(* CODESYS project bargeControl
   Author: Sigurd Rød Brekk
   Company: ScaleAQ
   Description: Control and monitoring of processe related to the barges.
   Title: bargeControl
   Version: 0.0.0

Project tree, tasks and I/O mapping:
  PFC100_Simulation : 750-8111 PFC100, WAGO, order no. 750-8111, version 6.2.0.1
    application Application
      libraries: Standard, 3.5.18.0 (System); WagoSysDynamicIoMapping, 1.0.4.0 (WAGO); SysTask, * (System)
      task BilgePump (cyclic, interval 100 ms, priority 1, watchdog 20 ms x 1) calls BilgePump
      task IOSimulation (cyclic, interval 100 ms, priority 1, watchdog 20 ms x 1) calls simulationMapping
      task TankLevel (cyclic, interval 100 ms, priority 1, watchdog 20 ms x 1) calls TankLevel
      GVL/
        global variables GVL_Simulation
      global variables PersistentVars
      program simulationMapping [ST]
      Symbols
    Kbus : Kbus, WAGO, version 2.1.0.1
        unmapped channels: K-BUS diagnostics
  SiteProgram : 750-8111 PFC100, WAGO, order no. 750-8111, version 6.2.0.1
    application Application
      libraries: Standard, 3.5.18.0 (System); WagoSysDynamicIoMapping, 1.0.4.0 (WAGO); SysTask, * (System)
      task BilgePump (cyclic, interval 100 ms, priority 2, watchdog 20 ms x 1) calls BilgePump
      task ReadIOCards (cyclic, interval 100 ms, priority 1, watchdog 20 ms x 1) calls DynamicIOConfig, ReadInputs
      task TankLevel (cyclic, interval 100 ms, priority 14, watchdog 20 ms x 1) calls TankLevel
      task WriteIOCards (cyclic, interval 100 ms, priority 15, watchdog 20 ms x 1) calls WriteOutputs
      GVL/
        global variables GVL_WagoIO
      global variables PersistentVars
      PRG/
        program DynamicIOConfig [ST]
        program ReadInputs [ST]
        program WriteOutputs [ST]
      Symbols
    Kbus : Kbus, WAGO, version 2.1.0.1
        unmapped channels: K-BUS diagnostics
  SoftSimulation : CODESYS Control Win V3 x64, 3S - Smart Software Solutions GmbH, version 3.5.19.50
    application Application
      libraries: Standard, 3.5.18.0 (System); SysTask, * (System)
      task BilgePump (cyclic, interval 100 ms, priority 1, watchdog 20 ms x 1) calls BilgePump
      task IOSimulation (cyclic, interval 100 ms, priority 1, watchdog 20 ms x 1) calls simulationMapping
      task TankLevel (cyclic, interval 100 ms, priority 1, watchdog 20 ms x 1) calls TankLevel
      task TrendRecordingTask (cyclic, interval 100 ms, priority 31) calls VisuTrendStorageAccess.GlobalInstances.g_TrendRecordingManager.CyclicCall
      task VISU_TASK (cyclic, interval 100 ms, priority 31) calls VisuElems.Visu_Prg
      global variables GVL_Simulation
      global variables PersistentVars
      program simulationMapping [ST]
      Symbols
      Trend Recording Manager
        TrendRecording
      visualisation Visualization
  ENUM/
    data type AlarmState
    data type powerState
    data type tankShape
    data type unitType
  FB/
    function block AlarmManagement [ST]
    function block BilgeControl [ST]
    function block Butterworth [ST]
  FUNCTION/
    function analogInputToMeter [ST]
    function heightToVolume [ST]
  text list GlobalTextList
  GVL/
    global variables GVL_IO
    global variables GVL_Retain
    global variables GVL_UPS
  PRG/
    program BilgePump [ST]
    program TankLevel [ST]
  STRUCT/
    data type AlarmStructBilge
    data type AlarmStructTankLevel
    data type BilgeObject
    data type IOSetup
    data type PowerSupply
    data type TankLevelObject
    data type UPS
*)

// ENUM/AlarmState
{attribute 'qualified_only'}
{attribute 'strict'}
TYPE AlarmState :
(
	Normal,
	UnacknowledgedAlarm,
	AcknowledgedAlarm,
	RTNunacknowledged
);
END_TYPE

// ENUM/powerState
{attribute 'qualified_only'}
{attribute 'strict'}
TYPE powerState :
(
	normal,
	noVoltage,
	fuseBlown
);
END_TYPE

// ENUM/tankShape
{attribute 'qualified_only'}
{attribute 'strict'}
TYPE tankShape :
(
	notDefined,
	rectangle,
	cylindrical
);
END_TYPE

// ENUM/unitType
{attribute 'qualified_only'}
{attribute 'strict'}
TYPE unitType :
(
	bar,
	meter
);
END_TYPE

// STRUCT/AlarmStructBilge
TYPE AlarmStructBilge :
STRUCT
	waterAlarmState				: AlarmState;
	acknowledgeWaterDetAlm		: BOOL;
	dieselAlarmState			: AlarmState;
	acknowledgeDieselDetAlm		: BOOL;
	manualStartAlarmState		: AlarmState;
	acknowledgeManualStartAlm	: BOOL;
END_STRUCT
END_TYPE

// STRUCT/AlarmStructTankLevel
TYPE AlarmStructTankLevel :
STRUCT
	LAL						: AlarmState;
	acknowledgeLAL			: BOOL;
	LAH						: AlarmState;
	acknowledgeLAH			: BOOL;
	outOfRange				: AlarmState;
	acknowledgeoutOfRange	: BOOL;
END_STRUCT
END_TYPE

// STRUCT/BilgeObject
TYPE BilgeObject :
STRUCT
	available				: BOOL;
	enable					: BOOL;
	auto					: BOOL;
	startManual				: BOOL;
	leakageDetected			: BOOL;
	dieselDetected			: BOOL;
	activateDieselDetection	: BOOL;
	startPump				: BOOL;
	Alarm					: AlarmStructBilge;
END_STRUCT
END_TYPE

// STRUCT/IOSetup
TYPE IOSetup :
STRUCT
	availableBilgeInputs	: INT;
	availableBilgeOutputs	: INT;
	availableAnalogInputs	: INT;
	IOFault					: BOOL;
END_STRUCT
END_TYPE

// STRUCT/PowerSupply
TYPE PowerSupply :
STRUCT
	available	: BOOL;
	state		: powerState;
END_STRUCT
END_TYPE

// STRUCT/TankLevelObject
TYPE TankLevelObject :
STRUCT
	available			: BOOL; //Checks if IO is available in K-BUS
	enable				: BOOL; //Enabled from SiteControl
	engRangeMin			: REAL; //Range on instrument [bar]
	engRangeMax 		: REAL; //Range on instrument [bar]
	rawInput 			: WORD; //input WORD from AD-converter
	filteredInput		: REAL; //filtered input WORD (low pass filter)
	density				: REAL; //density for liquid [kg/m^3]
	levelHeightOuput	: REAL; //height of liquid column [m]
	levelVolumeOutput	: REAL; //Volume [litre]
	tankShape			: tankShape;
	tankparameter		: ARRAY [1..2] OF REAL;
	SetPointLAL			: REAL; //[m]
	SetPointLAH			: REAL; //[m]
	Alarm				: AlarmStructTankLevel;
END_STRUCT
END_TYPE

// STRUCT/UPS
TYPE UPS :
STRUCT
	batteryHealthy	: BOOL;
	mainsConnected	: BOOL;
END_STRUCT
END_TYPE

// GVL/GVL_IO
{attribute 'qualified_only'}
VAR_GLOBAL	
	availableIO			: IOSetup;
END_VAR

// GVL/GVL_Retain
{attribute 'qualified_only'}
VAR_GLOBAL PERSISTENT RETAIN
	bilgePumpArray	: ARRAY [1..28] OF BilgeObject;
	tankLevelArray		: ARRAY [1..12] OF TankLevelObject;
END_VAR

// GVL/GVL_UPS
{attribute 'qualified_only'}
VAR_GLOBAL
	ups : UPS;
END_VAR

// PFC100_Simulation/Application/PersistentVars
{attribute 'qualified_only'}
VAR_GLOBAL PERSISTENT RETAIN
	// Generated instance path of persistent variable
	__POOL.GVL_Retain.bilgePumpArray: ARRAY [1..28] OF BilgeObject;
	// Generated instance path of persistent variable
	__POOL.GVL_Retain.tankLevelArray: ARRAY [1..12] OF TankLevelObject;
END_VAR

// SiteProgram/Application/PersistentVars
{attribute 'qualified_only'}
VAR_GLOBAL PERSISTENT RETAIN
	// Generated instance path of persistent variable
	__POOL.GVL_Retain.bilgePumpArray: ARRAY [1..28] OF BilgeObject;
	// Generated instance path of persistent variable
	__POOL.GVL_Retain.tankLevelArray: ARRAY [1..12] OF TankLevelObject;
END_VAR

// SoftSimulation/Application/GVL_Simulation
{attribute 'qualified_only'}
VAR_GLOBAL
tankLevelSim	: ARRAY [1..12] OF WORD;
bilgeLimitSwitch	: ARRAY [1..28] OF BOOL;
bilgePumpStart		: ARRAY [1..28] OF BOOL;
END_VAR

// SoftSimulation/Application/PersistentVars
{attribute 'qualified_only'}
VAR_GLOBAL PERSISTENT RETAIN
	// Generated instance path of persistent variable
	__POOL.GVL_Retain.bilgePumpArray: ARRAY [1..28] OF BilgeObject;
	// Generated instance path of persistent variable
	__POOL.GVL_Retain.tankLevelArray: ARRAY [1..12] OF TankLevelObject;
END_VAR

// PFC100_Simulation/Application/GVL/GVL_Simulation
{attribute 'qualified_only'}
VAR_GLOBAL
tankLevelSim	: ARRAY [1..12] OF WORD;
bilgeLimitSwitch	: ARRAY [1..28] OF BOOL;
bilgePumpStart		: ARRAY [1..28] OF BOOL;
END_VAR

// SiteProgram/Application/GVL/GVL_WagoIO
{attribute 'qualified_only'}
VAR_GLOBAL
	digitalInputCollection	: ARRAY [1..3] OF WagoSysDynamicIoMapping.I_Module;
	digitalOutputCollection	: ARRAY [1..3] OF WagoSysDynamicIoMapping.I_Module;
	analogInputCollection	: ARRAY [1..3] OF WagoSysDynamicIoMapping.I_Module;
	
END_VAR

// PRG/BilgePump
PROGRAM BilgePump
VAR
	i	: INT;
	BilgeControlArray	: ARRAY[1..28] OF BilgeControl;
	BilgeAlarm			: ARRAY[1..28] OF AlarmManagement;
END_VAR

FOR i := 1 TO 28 DO 
	IF (GVL_Retain.bilgePumpArray[i].available AND GVL_Retain.bilgePumpArray[i].enable) THEN
		BilgeControlArray[i](
			//INPUTS
			leakageDetected			:= GVL_Retain.bilgePumpArray[i].leakageDetected,
			dieselDetected			:= GVL_Retain.bilgePumpArray[i].dieselDetected,
			activateDieselDetection	:= GVL_Retain.bilgePumpArray[i].activateDieselDetection,
			auto					:= GVL_Retain.bilgePumpArray[i].auto,
			startManual				:= GVL_Retain.bilgePumpArray[i].startManual,
			
			//OUTPUTS
			startPump				=> GVL_Retain.bilgePumpArray[i].startPump
		);
		
		//Alarm management	
		//Alarm state for water detection
		BilgeAlarm[i](
			AbnormalCondition		:= GVL_Retain.bilgePumpArray[i].leakageDetected,
			Acknowledge				:= GVL_Retain.bilgePumpArray[i].Alarm.acknowledgeWaterDetAlm,
			ProcessAlarmState		:= GVL_Retain.bilgePumpArray[i].Alarm.waterAlarmState,
		);
		//Alarm state for disel detection
		BilgeAlarm[i](
			AbnormalCondition		:= GVL_Retain.bilgePumpArray[i].dieselDetected,
			Acknowledge				:= GVL_Retain.bilgePumpArray[i].Alarm.acknowledgeDieselDetAlm,
			ProcessAlarmState		:= GVL_Retain.bilgePumpArray[i].Alarm.dieselAlarmState,
		);
		//Alarm state for manual start
		BilgeAlarm[i](
			AbnormalCondition		:= GVL_Retain.bilgePumpArray[i].startManual,
			Acknowledge				:= GVL_Retain.bilgePumpArray[i].Alarm.acknowledgeManualStartAlm,
			ProcessAlarmState		:= GVL_Retain.bilgePumpArray[i].Alarm.manualStartAlarmState,
		);
	ELSE
		GVL_Retain.bilgePumpArray[i].startPump := FALSE;
	END_IF
END_FOR

END_PROGRAM

// FB/BilgeControl
FUNCTION_BLOCK BilgeControl
VAR_INPUT
	leakageDetected			: BOOL;
	dieselDetected			: BOOL;
	activateDieselDetection	: BOOL;
	auto					: BOOL;
	startManual				: BOOL;
END_VAR
VAR_OUTPUT
	startPump				: BOOL;
END_VAR
VAR
	pumpHysteresis	:	TOF;
END_VAR

IF auto THEN
	pumpHysteresis(IN := leakageDetected,PT := T#60S);
	IF (NOT(activateDieselDetection AND dieselDetected) AND leakageDetected) THEN // Only activate bilge pump if diesel is not detected (while activated).
		startPump := pumpHysteresis.Q;
	ELSE 
		startPump := FALSE;
	END_IF
ELSE
	IF startManual THEN
		startPump := TRUE;
	ELSE
		startPump := FALSE;
	END_IF
END_IF

END_FUNCTION_BLOCK

// FB/AlarmManagement
FUNCTION_BLOCK AlarmManagement
VAR_INPUT
	AbnormalCondition	: BOOL;
	Acknowledge			: BOOL;
END_VAR
VAR_IN_OUT
	ProcessAlarmState			: AlarmState;
END_VAR

CASE ProcessAlarmState OF
			0:
				//NORMAL OPERATION
				IF AbnormalCondition THEN
					ProcessAlarmState := 1;
				END_IF
			1:
				//UNACKNOWLEDGED ALARM
				IF NOT AbnormalCondition THEN
					ProcessAlarmState := 3;
				END_IF
				IF Acknowledge THEN
					ProcessAlarmState := 2;
				END_IF
			2:	
				//ACKNOWLEDGED ALARM
				IF NOT AbnormalCondition THEN
					ProcessAlarmState := 0;
				END_IF
			3:
			
				//RTN unacknowledged
				IF AbnormalCondition THEN
					ProcessAlarmState := 1;
				END_IF
				IF Acknowledge THEN
					ProcessAlarmState := 0;
				END_IF
		END_CASE

END_FUNCTION_BLOCK

// PFC100_Simulation/Application/simulationMapping
PROGRAM simulationMapping
VAR
	i	: INT;
	filter				: ARRAY[1..12] OF Butterworth; // second order butterworth filter 
END_VAR

//READ DIGITAL INPUTS FROM IO-CARD
FOR i := 1 TO 28 DO 
	IF (GVL_Retain.bilgePumpArray[i].available AND GVL_Retain.bilgePumpArray[i].enable) THEN
		GVL_Retain.bilgePumpArray[i].leakageDetected := GVL_Simulation.bilgeLimitSwitch[i];
	END_IF
END_FOR

FOR i	:= 1 TO 12 DO
	IF (GVL_Retain.tankLevelArray[i].available AND GVL_Retain.tankLevelArray[i].enable) THEN
	GVL_Retain.tankLevelArray[i].rawInput := GVL_Simulation.tankLevelSim[i];
	//Filter input signal
	filter[i](fc := 0.01, u_in:= GVL_Retain.tankLevelArray[i].rawInput, y_out => GVL_Retain.tankLevelArray[i].filteredInput);
	END_IF
END_FOR

IF (GVL_Retain.bilgePumpArray[i].available AND GVL_Retain.bilgePumpArray[i].enable) THEN
	GVL_Simulation.bilgePumpStart[i] := GVL_Retain.bilgePumpArray[i].startPump;
END_IF

END_PROGRAM

// SoftSimulation/Application/simulationMapping
PROGRAM simulationMapping
VAR
	i	: INT;
	filter				: ARRAY[1..12] OF Butterworth; // second order butterworth filter 
END_VAR

//READ DIGITAL INPUTS FROM IO-CARD
FOR i := 1 TO 28 DO 
	IF (GVL_Retain.bilgePumpArray[i].available AND GVL_Retain.bilgePumpArray[i].enable) THEN
		GVL_Retain.bilgePumpArray[i].leakageDetected := GVL_Simulation.bilgeLimitSwitch[i];
	END_IF
END_FOR

FOR i	:= 1 TO 12 DO
	IF (GVL_Retain.tankLevelArray[i].available AND GVL_Retain.tankLevelArray[i].enable) THEN
	GVL_Retain.tankLevelArray[i].rawInput := GVL_Simulation.tankLevelSim[i];
	//Filter input signal
	filter[i](fc := 0.01, u_in:= GVL_Retain.tankLevelArray[i].rawInput, y_out => GVL_Retain.tankLevelArray[i].filteredInput);
	END_IF
END_FOR

IF (GVL_Retain.bilgePumpArray[i].available AND GVL_Retain.bilgePumpArray[i].enable) THEN
	GVL_Simulation.bilgePumpStart[i] := GVL_Retain.bilgePumpArray[i].startPump;
END_IF

END_PROGRAM

// FB/Butterworth
FUNCTION_BLOCK Butterworth
VAR_INPUT
	fc		: REAL; //cut-off frequency
	u_in	: WORD; //filter input
END_VAR
VAR_OUTPUT
	y_out	: REAL; //filter output
END_VAR
VAR
	yk		: REAL := 0;
	ykm1	: REAL := 0;
	ykm2	: REAL := 0;
	uk		: REAL := 0;
	ukm1	: REAL	:= 0;
	ukm2	: REAL	:= 0;
	//TEST
	hTask:       SysTask.RTS_IEC_HANDLE; // task handle
	Tsu		: UDINT; // interval in micro seconds
	fsample		: REAL;
	fs			: REAL;
	
	A_2		: REAL;
	B_0		: REAL;
	B_1		: REAL;
	B_2		: REAL;
	
	N0		: REAL;
	N1		: REAL;
	N2		: REAL;
	D0		: REAL;
	D1		: REAL;
	D2		: REAL;
END_VAR

SysTaskGetCurrent(ADR(hTask));
SysTaskGetInterval(hTask, Tsu);
fsample := 1000000/(UDINT_TO_REAL(Tsu));
fs := 2*TAN(3.1415926536*((fc)/(fsample)));


uk 		:= WORD_TO_REAL(u_in);

A_2 := LREAL_TO_REAL(EXPT(2*3.1415926536*fs,2));
B_0 := 1;
B_1 := LREAL_TO_REAL(SQRT(2));
B_2 := A_2;

N0 := A_2;
N1 := 2*(A_2);
N2 := A_2;
D0 := B_2 + 2*fs*B_1 + 4*LREAL_TO_REAL(EXPT(fs,2))*B_0;
D1 := 2*(B_2 - 4*LREAL_TO_REAL(EXPT(fs,2))*B_0);
D2 := B_2 - 2*fs*B_1 + 4*LREAL_TO_REAL(EXPT(fs,2))*B_0;




yk		:= ((((N0)/(D0))/1) * (1*uk + ((N1)/(N0))*ukm1 + ((N2)/(N0))*ukm2)) - ((((D1)/(D0))*ykm1+((D2)/(D0))*ykm2));

ykm2 	:= ykm1;
ykm1 	:= yk;

ukm2	:= ukm1;
ukm1	:= uk;

y_out 	:= WORD_TO_REAL(REAL_TO_WORD(yk));

END_FUNCTION_BLOCK

// PRG/TankLevel

PROGRAM TankLevel
VAR
	i	: INT;
	TankAlarm			: ARRAY[1..12] OF AlarmManagement;

	//Alarm conditions
	fluidHigh			: BOOL;
	fluidLow			: BOOL;
	signalFault			: BOOL;
	
END_VAR

FOR i := 1 TO 12 DO 
	IF (GVL_Retain.tankLevelArray[i].available AND GVL_Retain.tankLevelArray[i].enable) THEN
		//Calculate level hegiht
		GVL_Retain.tankLevelArray[i].levelHeightOuput := analogInputToMeter(
			fluidDensity	:= GVL_Retain.tankLevelArray[i].density,
			engRangeMin		:= GVL_Retain.tankLevelArray[i].engRangeMin,
			engRangeMax		:= GVL_Retain.tankLevelArray[i].engRangeMax,
			input			:= GVL_Retain.tankLevelArray[i].filteredInput
		);
		//CALCULATE VOLUME IF DEFINED
		GVL_Retain.tankLevelArray[i].levelVolumeOutput := heightToVolume(
			GVL_Retain.tankLevelArray[i].levelHeightOuput,
			GVL_Retain.tankLevelArray[i].tankShape, 
			GVL_Retain.tankLevelArray[i].tankparameter);
		
		//CHECK IF LEVEL IS BELOW SET POINT FOR LAL
		IF (GVL_Retain.tankLevelArray[i].levelHeightOuput < GVL_Retain.tankLevelArray[i].SetPointLAL) AND (GVL_Retain.tankLevelArray[i].SetPointLAL > 0)  THEN
			fluidLow := TRUE;
		ELSE
			fluidLow := FALSE;
		END_IF
		//CHECK IF LEVEL IS ABOVE SET POINT FOR LAH
		IF (GVL_Retain.tankLevelArray[i].levelHeightOuput > GVL_Retain.tankLevelArray[i].SetPointLAH) AND (GVL_Retain.tankLevelArray[i].SetPointLAH > 0)  THEN
			fluidHigh := TRUE;
		ELSE
			fluidHigh := FALSE;
		END_IF
		//CHECK IF TRANSMITTER VALUE IS OUT OF RANGE - Analog input gives the value 3 if the current is < 3mA, and 32767 if current > 21mA
		IF (GVL_Retain.tankLevelArray[i].rawInput = 3) OR (GVL_Retain.tankLevelArray[i].rawInput = 32767)  THEN
			signalFault := TRUE;
		ELSE
			signalFault := FALSE;
		END_IF
		
		//ALARM MANAGEMENT
		//Alarm state for low level
		TankAlarm[i](
			AbnormalCondition		:= fluidLow,
			Acknowledge				:= GVL_Retain.tankLevelArray[i].Alarm.acknowledgeLAL,
			ProcessAlarmState		:= GVL_Retain.tankLevelArray[i].Alarm.LAL
		);
		//Alarm state for high level
		TankAlarm[i](
			AbnormalCondition		:= fluidHigh,
			Acknowledge				:= GVL_Retain.tankLevelArray[i].Alarm.acknowledgeLAH,
			ProcessAlarmState		:= GVL_Retain.tankLevelArray[i].Alarm.LAH
		);
		//Alarm state for transmitter out of range
		TankAlarm[i](
			AbnormalCondition		:= signalFault,
			Acknowledge				:= GVL_Retain.tankLevelArray[i].Alarm.acknowledgeoutOfRange,
			ProcessAlarmState		:= GVL_Retain.tankLevelArray[i].Alarm.outOfRange
		);
	END_IF
END_FOR

END_PROGRAM

// FUNCTION/analogInputToMeter
FUNCTION analogInputToMeter : REAL //in meters
VAR_INPUT
	fluidDensity		: REAL; //kg/m^3
	engRangeMin			: REAL; // bar
	engRangeMax			: REAL; // bar
	input				: REAL;
END_VAR
VAR
	g					: REAL := 9.8; //[m/s^2]
	res					: REAL := 4095;//analog input resolution
END_VAR

//h = (P)/(rho * g)
IF (fluidDensity > 0) THEN
	analogInputToMeter := ((input*(engRangeMax-engRangeMin)/res)*100000)/(fluidDensity*g);
ELSE
	 analogInputToMeter := 0;
END_IF

END_FUNCTION

// FUNCTION/heightToVolume
FUNCTION heightToVolume : REAL
VAR_INPUT
	height		: REAL;
	shape		: tankShape;
	parameters	: ARRAY [1..2] OF REAL;
END_VAR
VAR
	pi	: REAL := 3.141592653589793238462;
END_VAR

CASE shape OF
			1:
				heightToVolume := parameters[1]*parameters[2]*height;
			2:	
				heightToVolume := pi*LREAL_TO_REAL(EXPT(parameters[1],2))*height;
		END_CASE

END_FUNCTION

// SiteProgram/Application/PRG/DynamicIOConfig
PROGRAM DynamicIOConfig
VAR
	coCollection 	: WagoSysDynamicIoMapping.I_Modules;
	bInput 	: BYTE;
	oStatus : WagoSysErrorBase.FbResult;
	//counter for looping through IO-modules and adding them in separate arrays
	i	: UINT;
	j	: INT;
	cnt1	: UINT	:= 0;
	cnt2	: UINT	:= 0;
	cnt3	: UINT	:= 0;

	//DEBUG
	testString	: STRING;
	
	//maximum limit for expected IO-modules.
	limitDigitalInputs	: INT	:= 3;
	limitDigitalOutputs	: INT	:= 3;
	limitAnalogInputs	: INT	:= 3;
	
	//start bit for sorting IO modules only upon first scan of program. Ommit this code when application is running.
	firstScan	:	BOOL := TRUE;
END_VAR


IF firstScan THEN
	coCollection := DynKbusIoManager.coModules;
	FOR i := 1 TO coCollection.uiModuleCount DO
		IF (FIND(coCollection.aIModules[i].sOrderNumber,'16_IN') > 0) AND (cnt1 <= limitDigitalInputs - 1) THEN
			cnt1 := cnt1+1;
			GVL_WagoIO.digitalInputCollection[cnt1] := coCollection.aIModules[i];
		END_IF
		
		IF (FIND(coCollection.aIModules[i].sOrderNumber,'16_OUT') > 0) AND (cnt1 <= limitDigitalOutputs - 1) THEN
			cnt2 := cnt2+1;
			GVL_WagoIO.digitalOutputCollection[cnt2] := coCollection.aIModules[i];
		END_IF
		
		IF (FIND(coCollection.aIModules[i].sOrderNumber,'750-0455') > 0) AND (cnt1 <= limitAnalogInputs - 1) THEN
			cnt3 := cnt3+1;
			GVL_WagoIO.analogInputCollection[cnt3] := coCollection.aIModules[i];
		END_IF
	END_FOR
	
	GVL_IO.availableIO.availableBilgeInputs := (16 * UINT_TO_INT(cnt1)) - 4; //Reserve four for dieseldet.
	GVL_IO.availableIO.availableBilgeOutputs := (16 * UINT_TO_INT(cnt2)) - 4;//Reserve four for hardwired alarm signals
	IF GVL_IO.availableIO.availableBilgeOutputs < 1 OR GVL_IO.availableIO.availableBilgeInputs < 1 THEN
		GVL_IO.availableIO.IOFault := TRUE; //Give IO fault if minimum required IO is not met.
	END_IF
	
	GVL_IO.availableIO.availableAnalogInputs := 4 * UINT_TO_INT(cnt3);
	
	FOR j := 1 TO GVL_IO.availableIO.availableBilgeOutputs DO 
		IF GVL_IO.availableIO.availableBilgeInputs >= j  THEN
			GVL_Retain.bilgePumpArray[j].available := TRUE;
		END_IF
	END_FOR
	
	FOR j := 1 TO GVL_IO.availableIO.availableAnalogInputs DO 
		GVL_Retain.tankLevelArray[j].available := TRUE;
	END_FOR

	firstScan := FALSE; //Only do this config during startup.
END_IF

END_PROGRAM

// SiteProgram/Application/PRG/ReadInputs
PROGRAM ReadInputs
VAR
	i	:	INT;
	j	: 	INT;
	
	filter				: ARRAY[1..12] OF Butterworth; // second order butterworth filter 
END_VAR

//READ DIGITAL INPUTS FROM IO-CARD (WAGO DYNAMIC IO LIBRARY) and sort them in ascendig order. 
FOR i := 1 TO 28 DO 
	IF (GVL_Retain.bilgePumpArray[i].available AND GVL_Retain.bilgePumpArray[i].enable) THEN
		GVL_Retain.bilgePumpArray[i].leakageDetected := GVL_WagoIO.digitalInputCollection[1+TRUNC((i-1)/16)].GetProcessInBit(
			DINT_TO_UINT(TRUNC(((i-1) MOD 16)/8)),
			((INT_TO_USINT(i-1) MOD 16) MOD 8));
		IF (i <= 4) THEN
			GVL_Retain.bilgePumpArray[i].dieselDetected := GVL_WagoIO.digitalInputCollection[(GVL_IO.availableIO.availableBilgeInputs + 4)/16].GetProcessInBit(
				1,
				INT_TO_USINT(i)+3);
		END_IF
	END_IF
END_FOR
		
//READ ANALOG INPUTS FROM IO-CARD (WAGO DYNAMIC IO LIBRARY) and sort them in ascendig order. 
FOR i := 1 TO 12 DO 
	IF (GVL_Retain.tankLevelArray[i].available AND GVL_Retain.tankLevelArray[i].enable) THEN
		//READ INPUT FROM IO-CARD
		GVL_Retain.tankLevelArray[i].rawInput := SHR(GVL_WagoIO.analogInputCollection[1+TRUNC((i-1)/4)].GetProcessInWord(
			INT_TO_UINT((i-1)*2)),
			4
			);
		//Filter input signal
		filter[i](fc := 0.01, u_in:= GVL_Retain.tankLevelArray[i].rawInput, y_out => GVL_Retain.tankLevelArray[i].filteredInput);
	END_IF
END_FOR

END_PROGRAM

// SiteProgram/Application/PRG/WriteOutputs
PROGRAM WriteOutputs
VAR
	i	: INT;
END_VAR

//WRITE DIGITAL OUTPUTS TO IO-CARD (WAGO DYNAMIC IO LIBRARY) in ascending order. 
FOR i := 1 TO 28 DO 
	IF (GVL_Retain.bilgePumpArray[i].available AND GVL_Retain.bilgePumpArray[i].enable) THEN
		GVL_WagoIO.digitalOutputCollection[1+TRUNC((i-1)/16)].SetProcessOutBit(
			DINT_TO_UINT(TRUNC(((i-1) MOD 16)/8)),
			((INT_TO_USINT(i-1) MOD 16) MOD 8),
			GVL_Retain.bilgePumpArray[i].startPump);
	END_IF	
END_FOR

END_PROGRAM

// SoftSimulation/Application/Visualization
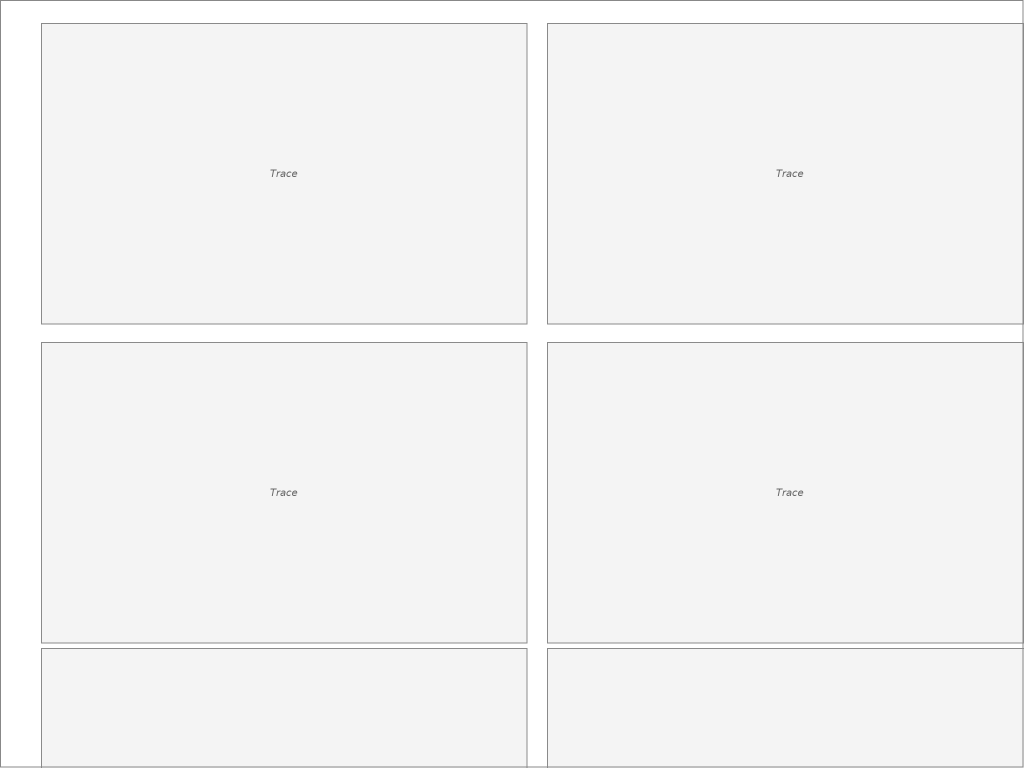
VISUALIZATION Visualization  // 1024x768
    Trace (41,23 486x301)
    Trace (547,23 486x301)
    Trace (1023,23 486x301)
    Trace (41,342 486x301)
    Trace (547,342 486x301)
    Trace (1023,342 486x301)
    Trace (547,648 486x301)
    Trace (41,648 486x301)
END_VISUALIZATION
